PROGRAM MAIN

VAR
	INTENSITY_BUTTON : INT;
	SUGAR_BUTTON : INT :=1;
	start : BOOL := FALSE;
	Tfill: TON;
	FILLING : BOOL := FALSE;
	WaterLevel : BOOL := FALSE;
	Level : REAL;
	Theat: TON;
    WaterTemp :REAL;
	HEATING : BOOL := FALSE;
	Tbrew: TON;
    WaterReady : BOOL := FALSE;
	BREWING : BOOL := FALSE;
    Tend: TON;
	
	CoffeeBrewed : BOOL := FALSE;
	Tready: TON;
	
	
	TIMER : TON;
	
	SugarMessage : STRING(30);
	
	state : status := status.START;

	Tstarting: Ton;
END_VAR

CASE state OF

    status.START:  //initialization and start the machine
        GVL.CoffeeReady := FALSE; 
        FILLING := FALSE;
        HEATING := FALSE;
        BREWING := FALSE;
        WaterLevel := FALSE;
        WaterReady := FALSE;
		SugarMessage := '';
		
		IF start THEN
		Tstarting(IN:=TRUE, PT:= T#2S);
            IF Tstarting.Q THEN
			state := status.LEVELCHECK; //check if the water is enough
			LogMessage(msg := 'Machine started', cleaning := FALSE, 2);// show the message in GVL of the current preparation state 
			Tstarting(IN:=FALSE);
			GVL.CoffeeReady:=FALSE;
			END_IF
        END_IF;       
	
    // over 80% is sufficient, otherwise the water has to be filled	
	status.LEVELCHECK: // over 80% is sufficient, otherwise the water has to be filled
	IF Level >= 80 THEN
		state := status.HEAT;
		WaterLevel := TRUE;
	ELSIF Level < 80 THEN
 		state:=status.FILL;
	END_IF
	
    //this status only if the water is under 80%
    status.FILL:  
		  Tfill(IN := TRUE, PT := T#8S);
		FILLING:= TRUE;
        FILLING := NOT WaterLevel; 
        WaterLevel := NOT FILLING;
        IF Tfill.Q THEN          
            Tfill(IN := FALSE);  
            FILLING := FALSE;    
            Level := 100;    
			LogMessage(msg := 'Water filled', cleaning := FALSE, 2);// show the message in GVL of the current preparation state 
            State := status.HEAT;              
        END_IF
		IF NOT start THEN
			state := status.START;
		END_IF
		
	//when the water is checked, the heating process starts
	status.HEAT:
        Theat (IN:=TRUE, PT := T#5S);
		HEATING := TRUE;
		HEATING := NOT WaterReady;
		WaterReady := NOT HEATING;

		IF Theat.Q THEN
			HEATING := FALSE;
			WaterTemp := 100;
			Level := Level - 10;
			Theat(IN:= FALSE);
			state := status.WATERREADY;
			LogMessage(msg := 'Water heating', cleaning := FALSE, 2);	// show the message in GVL of the current preparation state 		
		END_IF
		
	// when the right temperature of the water is reached, water is ready 
     status.WATERREADY:
	    WaterReady := TRUE;
        Theat(IN := TRUE, PT := T#5S);
        IF Theat.Q THEN
            WaterReady := FALSE;
            Theat(IN := FALSE);
			WaterTemp := 30;
            state := status.INTENSITY;
			LogMessage(msg := 'Water ready', cleaning := FALSE, 2); // show the message in GVL of the current preparation state
        END_IF
	// need to choose the intensity of the coffee, level 1 if the user wants light coffe and 3 if strong coffee
    status.INTENSITY:  
		 WaterLevel := FALSE;
         CASE INTENSITY_BUTTON OF
            1: Tbrew(IN := TRUE, PT := T#3S);
            2: Tbrew(IN := TRUE, PT := T#6S);
            3: Tbrew(IN := TRUE, PT := T#9S);
        ELSE
            Tbrew(IN := TRUE, PT := T#6S);  
        END_CASE
        BREWING := TRUE;  
		
        Tbrew (IN:=TRUE, PT:= T#5S);
        IF Tbrew.Q THEN
            BREWING := FALSE;     
            Tbrew(IN := FALSE); 
            State := status.SUGAR;  
            CoffeeBrewed := TRUE; 
			LogMessage(msg := 'water brewed', cleaning := FALSE, 2); // show the message in GVL of the current preparation state 
        END_IF
		
	// the user can choose the sugar quantity
    status.SUGAR: 
		IF CoffeeBrewed := TRUE THEN
		
		CASE SUGAR_BUTTON OF
			1: SugarMessage := 'no sugar';
			2: SugarMessage := 'medium sugar';
			3: SugarMessage := 'full sugar';
		ELSE
            SugarMessage := 'invalid selection';
		END_CASE
		state := status.READY;
	END_IF
	//The coffee is ready
    status.READY:  
        Tready(IN := TRUE, PT := T#2S);
        IF Tready.Q THEN
            Tready(IN := FALSE);
            state := status.END;
            start := FALSE;
			CoffeeBrewed := FALSE;
			GVL.CoffeeReady := TRUE;
			LogMessage(msg := 'Coffee ready', cleaning := FALSE, 2);// show the message in GVL of the current preparation state 
        END_IF
	
		
	// coffee is ready, step to visualize the message 'water ready' and wait the constumer grab the coffee
	status.END:  
        
        IF GVL.CLEANING THEN 
		  state:=status.CLEAN;
		  start := FALSE;
		  LogMessage(msg := 'Coffee ready', cleaning := TRUE, 2);// show the message in GVL of the current preparation state				
		ELSE 
            	
				start := FALSE;
				state := status.START;
			END_IF
        
		
	//waiting time to allow the machine cleaning program, if we reached 5 cycles
	status.CLEAN:
		 GVL.Tclean(IN:=TRUE, PT := T#10S);
		 IF GVL.Tclean.Q THEN
			 GVL.Tclean(IN:=FALSE);
			 state:=status.START;
			 LogMessage(msg := 'cleaned',cleaning := FALSE, 2);// show the message in GVL of the current preparation state
		 END_IF	  

END_CASE;

END_PROGRAM

(* stored: Version 1.1.0.1, ProductVersion 3.1.4024.15
   POU MAIN: Id {de3beb21-c81c-41bb-870c-964d49ad45d1}, SpecialFunc None *)
